FUNCTION_BLOCK "STD_LineSecStdSub2"	// FB 90
TITLE = Line and section control standard subroutines
//OPYRIGHT:    (C) 2000 BY  BUHLER LTD.
//                           CH-9240 UZWIL  SWITZERLAND
//
//PRODUCT:      STD_MU664    
//
//TITLE:        Line and section control standard subroutines
//              
//              Standardfunktionen für Linien und Sektionen              
//              
//
//--------------------------------------------------------------------------------
//
//IDENT:        AUTOR:              DEPT:                              DATE:
//
//STD_FB90.2.5  A. Egli             CT3                               11-Aug-2003
//              Sub2071: PICFU.SectionInfoCode     
//STD_FB90.2.4  Ph. Engler          MU664                             04-Aug-2003
//              Sub1061: LB not LW                    
//STD_FB90.2.3  Ph. Engler          MU664                             30-Aug-2003
//              Sub1061: Copy  #VarTemp.InOutValue3 to TmpDInt
//                       LB not LW                    
//STD_FB90.2.1  A.Egli              CT3                               14-Mai-2003
//              Sub1001: On Off Command Line
//STD_FB90.2.0  A.Egli              CT3                               18-Oct-2002
//              New release: Function moved from FC120 to FB90
//STD_FC120.1.12Ph. Engler          MU664                             23-Aug-2002
//              - Function (4,1) added: Search group manual mode
//STD_FC120.1.11Ph. Engler          MU664                              30-Apr-2002
//              - Function (1,55) and (2,55) modified: Stopping/Stopped
//STD_FC120.1.10Ph. Engler          MU664                              21-Mar-2002
//              - Function (2,55): starting until S.ToSSW.infStarted
//STD_FC120.1.9 Ph. Engler          MU664                              12-Mar-2002
//              Status codes for WinCoS implemented:
//              - General group colour code
//              - Line and Section info code
//STD_FC120.1.8 Ph. Engler          MU664                              20-Mar-2001
//              Line status colour for 2-4 section implemented
//STD_FC120.1.7 Ph. Engler          MU664                              20-Dec-2000
//              Pre stop weight for cmdSequenceStop
//STD_FC120.1.6 Ph. Engler          MU664                              14-Dec-2000
//              - Substitude BtmpInCode into recipe extended, tmpInCode 3 
//              - JS Job paramter flags (2,2) Sta-Address corrected
//STD_FC120.1.5 Ph. Engler          MU664                              01-Nov-2000
//              CmdSequenceStop only if section is in StActive           
//STD_FC120.1.4 Ph. Engler          MU664                              19-Okt-2000
//              Update SND-Binlist staSameSndRcv:
//               Suppression of the error meassage 'bin not found'
//STD_FC120.1.3 Ph. Engler          MU664                              28-Jun-2000
//              Section text and colour code extension 
//              with code 702, 703 and 1402
//STD_FC120.1.2 Ph. Engler          MU664                              04-May-2000
//              LS Line state/fault protocolling (1,10)
//               esXXX corrected 
//STD_FC120.1.1 Ph. Engler          MU664                              29-Mar-2000
//              Line log messages implemented
//STD_FC120.1.0 Ph. Engler          MU664                              05-Jan-2000
//              1st Release
//
//--------------------------------------------------------------------------------
//
//PURPOSE:      
//
//RESTRICTIONS:
//
//--------------------------------------------------------------------------------
//
AUTHOR : EA
FAMILY : STD
NAME : STD_FB90
VERSION : 2.5
VAR_INPUT
  InCode : INT ;
END_VAR
VAR
  Para : STRUCT
   ParSecNr : INT  := 1;
   ParLineDB_ParFirstSecDB : INT  := 320;
   spare4 : INT ;
   ParNextSecDB : INT ;	//Next section DB of this project line
   ParSecDataFirstByte : INT  := 240;
   ParSecDataLenNomValue : INT  := 20;
   ParSecDataLenAcValue : INT  := 20;
   ParBinDataFirstByte : INT  := 300;
   ParBinDataLength : INT  := 72;
  END_STRUCT ;
  VarTemp : STRUCT
   InOutValue1 : INT ;
   InOutValue2 : INT ;
   InOutValue3 : DINT ;
   InOutValue4 : DINT ;
   InOutValue5 : DINT ;
   InOutValue6 : DINT ;
  END_STRUCT ;
  ChangeBit : STRUCT
   spare : BYTE ;
   CBit1 : BOOL ;
   CBit2 : BOOL ;
   CBit3 : BOOL ;
   CBit4 : BOOL ;
  END_STRUCT ;
  ToASW : STRUCT
   spare00 : WORD ;
   CmdModify : BOOL ;
   CmdNewBatch : BOOL ;
   CmdDataMoved : BOOL ;
   InfSameJobPrevSec : BOOL ;
   InfSameJobNextSec : BOOL ;
   InfSameBatchPrevSec : BOOL ;
   InfSameBatchNextSec : BOOL ;
   InfSameJobLineDB : BOOL ;	//Job in reveive box is equal
   InfEmptyingTimeEnd : BOOL ;
   InfWayAdjustTimeEnd : BOOL ;
   spare32 : BOOL ;
   spare33 : BOOL ;
   spare34 : BOOL ;
   spare35 : BOOL ;
   spare36 : BOOL ;
   InfDataReady : BOOL ;
   Func : UDT 10601;
   Transition : STRUCT
    spare00 : BYTE ;
    ToPassive : BOOL ;
    ToWait : BOOL ;
    ToActive : BOOL ;
    ToReady : BOOL ;
    ToEmptying : BOOL ;
    ToEmptied : BOOL ;
    ToIdling : BOOL ;
   END_STRUCT ;
   spare10 : WORD ;
   spare12 : DWORD ;
   spare16 : DWORD ;
  END_STRUCT ;
  ToSSW : STRUCT
   InfStopped : BOOL ;
   spare01 : BOOL ;
   InfStarted : BOOL ;
   spare03 : BOOL ;
   spare04 : BOOL ;
   InfFeeding : BOOL ;
   spare06 : BOOL ;
   spare07 : BOOL ;
   spare00 : BOOL ;
   CmdGotoActive : BOOL ;
   CmdGotoReady : BOOL ;
   CmdGotoEmptying : BOOL ;
   CmdGotoEmptied : BOOL ;
   CmdGotoIdling : BOOL ;
   CmdGotoPassive : BOOL ;
   spare17 : BOOL ;
   InfReadyForNewBatch : BOOL ;
   CmdSendResult : BOOL ;
   InfPulseTimer : BOOL ;
   CmdNewWay : BOOL ;
   spare24 : BOOL ;
   spare25 : BOOL ;
   spare26 : BOOL ;
   InfReleaseEmptyingTime : BOOL ;
   Func : UDT 10601;
   InPrevSecDB : INT ;	//Previouse section DB in product flow
   InNextSecDB : INT ;	//Next section DB in product flow
   spare12 : DWORD ;
   spare16 : DWORD ;
  END_STRUCT ;
  PCWrite : STRUCT 	//PC Write : Section Data
   Hsk : STRUCT
    Q_Status : BOOL ;
    Q_Result : BOOL ;
    spare02 : BOOL ;
    spare03 : BOOL ;
    spare04 : BOOL ;
    spare05 : BOOL ;
    Q_MDEEData : BOOL ;	//Acknowledge data sended to MDEE by PCC
    Q_MYRAData : BOOL ;	//Acknowledge data sended to MYRA by PCC
    F_Define : BOOL ;
   END_STRUCT ;
   spare2 : WORD ;
   Func : UDT 10601;
   Value1 : INT ;
   Value2 : INT ;
   Value3 : INT ;
   ParWayAdjustTime : INT  := 2;
   Value5 : INT ;
   ParEmptyingTime : INT  := 20;
  END_STRUCT ;
  PCRead : STRUCT 	//PC Read : Section Data
   Hsk : STRUCT
    F_Status : BOOL ;
    F_Result : BOOL ;
    F_2 : BOOL ;
    F_3 : BOOL ;
    F_4 : BOOL ;
    F_5 : BOOL ;
    F_MDEEData : BOOL ;	//Request PCC to send data to MDEE
    F_MYRAData : BOOL ;	//Request PCC to send data to MYRA
   END_STRUCT ;
   ErrElement : INT ;
   ErrCode : INT ;
   ErrObject : INT ;	//(*new*)
   Step : STRUCT
    spare : BYTE ;
    StPassive : BOOL ;
    StWait : BOOL ;
    StActive : BOOL ;
    StReady : BOOL ;	//Line= Idling
    StEmptying : BOOL ;
    StEmptied : BOOL ;
    StIdling : BOOL ;
   END_STRUCT ;
   State : STRUCT
    spare : BYTE ;
    StStopped : BOOL ;
    StStarting : BOOL ;
    StStarted : BOOL ;
    StStopping : BOOL ;
    spare04 : BOOL ;
    StFeeding : BOOL ;
   END_STRUCT ;
   Fault : UDT 10602;
   Status : UDT 10603;
   StateColor : INT ;
   StateInfoCode : INT ;	//Line: GenGrpColorCode
   ExtStatus : INT ;
   OutWayAdjustTime_ExtOn : INT ;
   OutStartWarningTime : INT ;	//Copy of Startwarning modul
   OutEmptyingTime : INT ;
   Value7 : INT ;
   Value8 : INT ;
   Value9 : INT ;
   Value10 : INT ;
   Value11 : INT ;
   Value12 : INT ;
   Value13 : INT ;
   Value14 : INT ;
   Value15 : INT ;
   Value16 : INT ;
   Value17 : INT ;
   Value18 : INT ;
   Value19 : INT ;
  END_STRUCT ;
  JobNom : STRUCT 	//PC Read: Job header: Nominal values
   JobNr : DINT ;
   JobWeight : DINT ;	//Total Job weight
   BatchNo : INT  := 10;	//Number of batch requested form PC
   ScaleUsed : ARRAY  [1 .. 64 ] OF BOOL ;
   RecipeNr : INT ;
   BatchWeight : DINT ;
   BatchMinPpm : INT ;	//Minimum batch size [0.1%]
   BatchMaxPpm : INT ;	//Maximum batch size [0.1%]
   BatchNoOffset : INT ;	//Batch number of first batch
   MixingTime : INT ;	//Mixing time
   JobChangeTime : INT ;	//Job change time
   FeedingTime : INT ;	//Feeding Time
   Value13 : INT ;
   Value14 : INT ;
  END_STRUCT ;
  JobAc : STRUCT 	//PC Read: Job header: Actual values
   StaBatch : STRUCT
    spare0 : BOOL ;
    spare1 : BOOL ;
    spare2 : BOOL ;
    spare3 : BOOL ;
    spare4 : BOOL ;
    spare5 : BOOL ;
    StaEmptyingBatch : BOOL ;
    StaScaleRecipeValid : BOOL ;
    StaErrBatch : BOOL ;
    StaHandAddReady : BOOL ;
    StaRegistrated : BOOL ;
    StaLastBatch : BOOL ;
    StaDone : BOOL ;
   END_STRUCT ;
   JobWeight : DINT ;
   BatchNo : INT ;
   BatchNoCal : INT ;
   BatchWeightTarget : DINT ;	//Calculated target batch weight
   BatchWeightActual : DINT ;	//Actual weight of all dosed ingredient
   BatchSizePpm : INT ;	//Calculated batch size [1/1000]
   BatchValue8 : INT ;
   BatchValue9 : INT ;
   MixingTime : INT ;	//Mixing time
   JobChangeTime : INT ;	//Job change time
   FeedingTime : INT ;	//Feeding Time
   RecipePlace : INT ;	//Actual recipe place
   Value16 : INT ;
   Value17 : INT ;
   Value18 : INT ;
   Value19 : INT ;
  END_STRUCT ;
END_VAR
VAR_TEMP
  TmpWord : WORD ;
  TmpInt : INT ;
  TmpDInt : DINT ;
  TmpBool : BOOL ;
  tmpLineStStopped : BOOL ;
  tmpLineStaAutostart : BOOL ;
  tmpLineInfFeeding : BOOL ;
  DB9SecArray : DWORD ;	//Address Pointer Section in DB9
  tmpSecDB : INT ;
  tmpAddrGrInterfaceSec : DINT ;	//Pointer to Interface in section DB
  tmpLineDB : INT ;
  tmpRelevantGroups : DINT ;
  tmpSec_GenGrpCoulorCode : STRUCT
   lightGrey : BOOL ;
   Bit1 : BOOL ;
   darkGreen : BOOL ;
   magenta : BOOL ;
   red : BOOL ;
  END_STRUCT ;
  tmpLin_GenGrpCoulorCode : STRUCT
   lightGrey : BOOL ;
   Bit1 : BOOL ;
   darkGreen : BOOL ;
   magenta : BOOL ;
   red : BOOL ;
  END_STRUCT ;
  tmpStateColorS1 : STRUCT
   white : BOOL ;
   yellow : BOOL ;
   blue : BOOL ;
   dark_green : BOOL ;
   green : BOOL ;
   light_green : BOOL ;
   mangenta : BOOL ;
   red : BOOL ;
   Bit8 : BOOL ;
   Bit9 : BOOL ;
   Bit10 : BOOL ;
   Bit11 : BOOL ;
   Bit12 : BOOL ;
   brown : BOOL ;
   orange : BOOL ;
   tuerkis : BOOL ;
  END_STRUCT ;
  tmpStateColorS2 : STRUCT
   white : BOOL ;
   yellow : BOOL ;
   blue : BOOL ;
   dark_green : BOOL ;
   green : BOOL ;
   light_green : BOOL ;
   mangenta : BOOL ;
   red : BOOL ;
   Bit8 : BOOL ;
   Bit9 : BOOL ;
   Bit10 : BOOL ;
   Bit11 : BOOL ;
   Bit12 : BOOL ;
   brown : BOOL ;
   orange : BOOL ;
   tuerkis : BOOL ;
  END_STRUCT ;
  tmpStateColorS3 : STRUCT
   white : BOOL ;
   yellow : BOOL ;
   blue : BOOL ;
   dark_green : BOOL ;
   green : BOOL ;
   light_green : BOOL ;
   mangenta : BOOL ;
   red : BOOL ;
   Bit8 : BOOL ;
   Bit9 : BOOL ;
   Bit10 : BOOL ;
   Bit11 : BOOL ;
   Bit12 : BOOL ;
   brown : BOOL ;
   orange : BOOL ;
   tuerkis : BOOL ;
  END_STRUCT ;
  tmpStateColorS4 : STRUCT
   white : BOOL ;
   yellow : BOOL ;
   blue : BOOL ;
   dark_green : BOOL ;
   green : BOOL ;
   light_green : BOOL ;
   mangenta : BOOL ;
   red : BOOL ;
   Bit8 : BOOL ;
   Bit9 : BOOL ;
   Bit10 : BOOL ;
   Bit11 : BOOL ;
   Bit12 : BOOL ;
   brown : BOOL ;
   orange : BOOL ;
   tuerkis : BOOL ;
  END_STRUCT ;
  tmpStateColorLine : STRUCT
   white : BOOL ;
   yellow : BOOL ;
   blue : BOOL ;
   dark_green : BOOL ;
   green : BOOL ;
   light_green : BOOL ;
   mangenta : BOOL ;
   red : BOOL ;
   Bit8 : BOOL ;
   Bit9 : BOOL ;
   Bit10 : BOOL ;
   Bit11 : BOOL ;
   Bit12 : BOOL ;
   brown : BOOL ;
   orange : BOOL ;
   tuerkis : BOOL ;
  END_STRUCT ;
  tmpUserState : STRUCT 	//PIC FU
   stEmptying : BOOL ;
   stEmptied : BOOL ;
   stIdling : BOOL ;
   stFault : BOOL ;
   stHand : BOOL ;
   stHold : BOOL ;
   stStep : BOOL ;
   spare : BOOL ;
   stPassiv : BOOL ;
   stWait : BOOL ;
   stStarting : BOOL ;
   stStarted : BOOL ;
   stStopping : BOOL ;
   stStopped : BOOL ;
   stFeeding : BOOL ;
   stReady : BOOL ;
  END_STRUCT ;
END_VAR
BEGIN
NETWORK
TITLE = Init
      LAR2  P##InCode;
      L     DINO;
      T     #tmpLineDB;
      T     #tmpSecDB;
NETWORK
TITLE = Sub1001: LS Line On Off Command
//Called by line controler subroutines, with opened L-DB
      L     #InCode;
      L     1001;
      <>I;
      JC    LS01;
      L     #PCWrite.Value1;	// PCWrite.ExtFuncOn 
      T     #PCRead.OutWayAdjustTime_ExtOn;
//-Update ExtStatus------------------------
      L     #PCRead.ExtStatus;	// ExtStatus
      L     #PCWrite.Value1;	// PCWrite.ExtFuncOn 
      OD;	// 
      L     #PCWrite.Value2;	// PCWrite.ExtFuncOff 
      INVD;	//  
      AD;	//  
      T     #PCRead.ExtStatus;	//->ExtStatus
//Reset on commands 
      L     0;
      T     #PCWrite.Value1;	// PCWrite.ExtFuncOn 
//Reset off commands 
      L     0;
      T     #PCWrite.Value2;	// PCWrite.ExtFuncOff 
      BEU;
LS01: NOP   0;
NETWORK
TITLE = Sub1010: LS Line state/fault protocolling
//Called by line controler subroutines, with opened L-DB
//
//Output: LineDB.VarTemp.InOutValue1 = LineMsg
      L     #InCode;
      L     1010;
      <>I;
      JC    LS00;
//-Init var---
      L     0;
      T     MW 2018;
//Read old value: PCRead.StateColor
      L     #PCRead.StateColor;
      LAR1  P##tmpStateColorS1;	// LineDB.PCRead.StateColor
      T     LW [AR1,P#0.0];	//-->tmpStateColorS1
//-Generate summary step---
      A     #tmpStateColorS1.tuerkis;	// 
      =     M 2019.3;	// --> LineMsg.suspended
      SET;
      S     M 2019.0;	// --> LineMsg.terminated
      S     M 2019.1;	// --> LineMsg.stopped
      R     M 2019.2;	// --> LineMsg.started
      R     M 2019.4;	// --> LineMsg.faulted
      R     M 2019.5;	// --> LineMsg.warning
      R     M 2018.0;	// --> LineMsg.SenderEmpty
      R     M 2018.3;	// --> LineMsg.allPreselectRcvFull
      R     M 2018.4;	// --> LineMsg.MachinesNotAvailable
      L     #Para.ParLineDB_ParFirstSecDB;	// Para.ParFirstSecDB   
LOOP: T     #tmpSecDB;
      OPN   DI [#tmpSecDB];
      AN    #PCRead.Step.StPassive;	// Section
      AN    #PCRead.Step.StIdling;	// Section
      R     M 2019.0;	// --> LineMsg.terminated
      AN    #PCRead.State.StStopped;	// Section
      ON    #PCRead.Status.StaImmediateStopASW;	// Section
      R     M 2019.1;	// --> LineMsg.stopped
      AN    #PCRead.Step.StPassive;	// Section
      AN    #PCRead.Step.StIdling;	// Section
      S     M 2019.2;	// --> LineMsg.started
      A     #PCRead.Fault.EsMech;	// Section
      AN    #PCRead.Step.StPassive;	// Section
      AN    #PCRead.Step.StIdling;	// Section
      S     M 2019.4;	// --> LineMsg.faulted
      A     #PCRead.Fault.EsWarning;	// Section
      AN    #PCRead.Step.StPassive;	// Section
      AN    #PCRead.Step.StIdling;	// Section
      S     M 2019.5;	// --> LineMsg.warning
      A     #PCRead.Fault.EsEmpty;	// Section
      AN    #PCRead.Step.StPassive;	// Section
      AN    #PCRead.Step.StIdling;	// Section
      S     M 2018.0;	// --> LineMsg.SenderEmpty
      A     #PCRead.Fault.EsFull;	// Section
      AN    #PCRead.Step.StPassive;	// Section
      AN    #PCRead.Step.StIdling;	// Section
      S     M 2018.3;	// --> LineMsg.allPreselectRcvFull
      A     #PCRead.Fault.EsWayConflict;	// Section
      AN    #PCRead.Step.StPassive;	// Section
      AN    #PCRead.Step.StIdling;	// Section
      S     M 2018.4;	// --> LineMsg.MachinesNotAvailable
//-Check next section---
      L     0;
      L     #Para.ParNextSecDB;	// Section
      <>I;
      JC    LOOP;
//-Return messages---
      OPN   DI [#tmpLineDB];
      L     MW 2018;	// LineMsg
      T     #VarTemp.InOutValue1;
      BEU;
LS00: NOP   0;
NETWORK
TITLE = Sub1051: C1 Line status colour for 1 section
//Called by line controler subroutines
      L     #InCode;
      L     1051;
      <>I;
      JC    C100;
//Init
      L     0;
      LAR1  P##tmpStateColorLine;
      T     LW [AR1,P#0.0];	//-->tmpStateColorLine
//Read state of section 1
      L     #Para.ParLineDB_ParFirstSecDB;
      T     #tmpSecDB;
      OPN   DI [#tmpSecDB];	// Call 1st section
      L     #PCRead.StateColor;	// Section
      LAR1  P##tmpStateColorS1;
      T     LW [AR1,P#0.0];	//-->tmpStateColorS1
//-Red----------------------------------
      A     #tmpStateColorS1.red;	// Section
      S     #tmpStateColorLine.red;
      JC    C101;
//-Magenta------------------------------
      A     #tmpStateColorS1.mangenta;	// Section
      S     #tmpStateColorLine.mangenta;
      JC    C101;
//-Turkis-------------------------------
      A     #tmpStateColorS1.tuerkis;	// Section
      S     #tmpStateColorLine.tuerkis;
      JC    C101;
//-Brown--------------------------------
      A     #tmpStateColorS1.brown;	// Section
      S     #tmpStateColorLine.brown;
      JC    C101;
//-Orange-------------------------------
      A     #tmpStateColorS1.orange;	// Section
      S     #tmpStateColorLine.orange;
      JC    C101;
//-Lightgreen---------------------------
      A     #tmpStateColorS1.light_green;	// Section
      S     #tmpStateColorLine.light_green;
      JC    C101;
//-Green--------------------------------
      A     #tmpStateColorS1.green;	// Section
      S     #tmpStateColorLine.green;
      JC    C101;
//-Darkgreen----------------------------
      A     #tmpStateColorS1.dark_green;	// Section
      S     #tmpStateColorLine.dark_green;
      JC    C101;
//-Yellow-------------------------------
      A     #tmpStateColorS1.yellow;	// Section
      S     #tmpStateColorLine.yellow;
      JC    C101;
//-Blue---------------------------------
      A     #tmpStateColorS1.blue;	// Section
      S     #tmpStateColorLine.blue;
      JC    C101;
//-White--------------------------------
      A     #tmpStateColorS1.white;	// Section
      S     #tmpStateColorLine.white;	//(default)
//-Data to PCC--------------------------
C101: OPN   DI [#tmpLineDB];
      LAR1  P##tmpStateColorLine;
      L     LW [AR1,P#0.0];	// tmpStateColorLine
      L     #PCRead.StateColor;	// LineDB
      ==I;	// 
      BEC;
      S     #ChangeBit.CBit1;	// LineDB
      TAK;
      T     #PCRead.StateColor;	// LineDB
      BEU;
C100: NOP   0;
NETWORK
TITLE = Sub1052: C2 Line status colour for 2 section
//Called by line controler subroutines
//
//Inputs :
// no
//Outputs:
// no
//
      L     #InCode;
      L     1052;
      <>I;
      JC    C200;
//Init
      L     0;
      LAR1  P##tmpStateColorLine;
      T     LW [AR1,P#0.0];	//-->tmpStateColorLine
//Read Status Section 1
      L     #Para.ParLineDB_ParFirstSecDB;
      T     #tmpSecDB;
      OPN   DI [#tmpSecDB];	// Call 1st section DB Para.ParFirstSecDB
      L     #PCRead.StateColor;	// Section
      LAR1  P##tmpStateColorS1;
      T     LW [AR1,P#0.0];	//-->tmpStateColorS1
//Read Status Section2
      L     #Para.ParNextSecDB;	// Section
      T     #tmpSecDB;
      OPN   DI [#tmpSecDB];	// Call next section DB Para.ParNextSecDB
      L     #PCRead.StateColor;	// Section
      LAR1  P##tmpStateColorS2;
      T     LW [AR1,P#0.0];	//-->tmpStateColorS2
      OPN   DI [#tmpLineDB];	// Call line DB .Para.ParLineDB
//-Red----------------------------------
      A     #tmpStateColorS1.red;
      O     #tmpStateColorS2.red;
      S     #tmpStateColorLine.red;
      JC    C201;
//-Magenta------------------------------
      A     #tmpStateColorS1.mangenta;
      O     #tmpStateColorS2.mangenta;
      S     #tmpStateColorLine.mangenta;
      JC    C201;
//-Turkis-------------------------------
      A     #tmpStateColorS1.tuerkis;
      O     #tmpStateColorS2.tuerkis;
      S     #tmpStateColorLine.tuerkis;
      JC    C201;
//-Brown--------------------------------
      A     #tmpStateColorS1.brown;
      O     #tmpStateColorS2.brown;
      S     #tmpStateColorLine.brown;
      JC    C201;
//-Orange-------------------------------
      A     #tmpStateColorS1.orange;
      O     #tmpStateColorS2.orange;
      S     #tmpStateColorLine.orange;
      JC    C201;
//-Lightgreen---------------------------
      A     #tmpStateColorS1.light_green;
      O     #tmpStateColorS2.light_green;
      S     #tmpStateColorLine.light_green;
      JC    C201;
//-Green--------------------------------
      A     #tmpStateColorS1.green;
      O     #tmpStateColorS2.green;
      S     #tmpStateColorLine.green;
      JC    C201;
//-Darkgreen----------------------------
      A     #tmpStateColorS1.dark_green;
      O     #tmpStateColorS2.dark_green;
      S     #tmpStateColorLine.dark_green;
      JC    C201;
//-Blue---------------------------------
      A     #tmpStateColorS1.blue;
      O     #tmpStateColorS2.blue;
      S     #tmpStateColorLine.blue;
      JC    C201;
//-Yellow-------------------------------
      A     #tmpStateColorS1.yellow;
      O     #tmpStateColorS2.yellow;
      S     #tmpStateColorLine.yellow;
      JC    C201;
//-White--------------------------------
      A     #tmpStateColorS1.white;
      A     #tmpStateColorS2.white;
      S     #tmpStateColorLine.white;	// (default)
//-Data to PCC--------------------------
C201: OPN   DI [#tmpLineDB];
      LAR1  P##tmpStateColorLine;
      L     LW [AR1,P#0.0];	// tmpStateColorLine
      L     #PCRead.StateColor;	// LineDB
      ==I;
      BEC;
      S     #ChangeBit.CBit1;	// LineDB
      TAK;
      T     #PCRead.StateColor;	// LineDB
      BEU;
C200: NOP   0;
NETWORK
TITLE = Sub1053: C3 Line status colour for 3 section
//Called by line controler subroutines
//
//Inputs :
// no
//Outputs:
// no
//
      L     #InCode;
      L     1053;
      <>I;
      JC    C300;
//Init
      L     0;
      LAR1  P##tmpStateColorLine;
      T     LW [AR1,P#0.0];	//-->tmpStateColorLine
//Read Status Section1
      L     #Para.ParLineDB_ParFirstSecDB;
      T     #tmpSecDB;
      OPN   DI [#tmpSecDB];	// Call 1st section DB Para.ParFirstSecDB
      L     #PCRead.StateColor;	// Section
      LAR1  P##tmpStateColorS1;
      T     LW [AR1,P#0.0];	//-->tmpStateColorS1
//Read Status Section2
      L     #Para.ParNextSecDB;	// Section
      T     #tmpSecDB;
      OPN   DI [#tmpSecDB];	// Call next section DB Para.ParNextSecDB
      L     #PCRead.StateColor;	// Section
      LAR1  P##tmpStateColorS2;
      T     LW [AR1,P#0.0];	//-->tmpStateColorS2
//Read Status Section3
      L     #Para.ParNextSecDB;	// Section
      T     #tmpSecDB;
      OPN   DI [#tmpSecDB];	// Call next section DB Para.ParNextSecDB
      L     #PCRead.StateColor;	// Section
      LAR1  P##tmpStateColorS3;
      T     LW [AR1,P#0.0];	//-->tmpStateColorS3
//-Red----------------------------------
      OPN   DI [#tmpLineDB];
      A     #tmpStateColorS1.red;
      O     #tmpStateColorS2.red;
      O     #tmpStateColorS3.red;
      S     #tmpStateColorLine.red;
      JC    C301;
//-Magenta------------------------------
      A     #tmpStateColorS1.mangenta;
      O     #tmpStateColorS2.mangenta;
      O     #tmpStateColorS3.mangenta;
      S     #tmpStateColorLine.mangenta;
      JC    C301;
//-Turkis-------------------------------
      A     #tmpStateColorS1.tuerkis;
      O     #tmpStateColorS2.tuerkis;
      O     #tmpStateColorS3.tuerkis;
      S     #tmpStateColorLine.tuerkis;
      JC    C301;
//-Brown--------------------------------
      A     #tmpStateColorS1.brown;
      O     #tmpStateColorS2.brown;
      O     #tmpStateColorS3.brown;
      S     #tmpStateColorLine.brown;
      JC    C301;
//-Orange-------------------------------
      A     #tmpStateColorS1.orange;
      O     #tmpStateColorS2.orange;
      O     #tmpStateColorS3.orange;
      S     #tmpStateColorLine.orange;
      JC    C301;
//-Lightgreen---------------------------
      A     #tmpStateColorS1.light_green;
      O     #tmpStateColorS2.light_green;
      O     #tmpStateColorS3.light_green;
      S     #tmpStateColorLine.light_green;
      JC    C301;
//-Green--------------------------------
      A     #tmpStateColorS1.green;
      O     #tmpStateColorS2.green;
      O     #tmpStateColorS3.green;
      AN    #tmpStateColorS2.dark_green;
      S     #tmpStateColorLine.green;
      JC    C301;
//-Darkgreen----------------------------
//      U     #tmpStateColorS1.dark_green
      A     #tmpStateColorS2.dark_green;
//      U     #tmpStateColorS3.dark_green
      S     #tmpStateColorLine.dark_green;
      JC    C301;
//-Blue---------------------------------
      A     #tmpStateColorS1.blue;
      O     #tmpStateColorS2.blue;
      O     #tmpStateColorS3.blue;
      S     #tmpStateColorLine.blue;
      JC    C301;
//-Yellow-------------------------------
//      U     #tmpStateColorS1.yellow
      A     #tmpStateColorS2.yellow;
//      U     #tmpStateColorS3.yellow
      S     #tmpStateColorLine.yellow;
      JC    C301;
//-White--------------------------------
//      U     #tmpStateColorS1.white
      A     #tmpStateColorS2.white;
      A     #tmpStateColorS3.white;
      S     #tmpStateColorLine.white;	// (default)
      JC    C301;
//-Data to PCC--------------------------
C301: OPN   DI [#tmpLineDB];
      LAR1  P##tmpStateColorLine;
      L     LW [AR1,P#0.0];	// tmpStateColorLine
      L     #PCRead.StateColor;	// LineDB
      ==I;	// 
      BEC;
      S     #ChangeBit.CBit1;	// LineDB
      TAK;
      T     #PCRead.StateColor;	// LineDB
      BEU;
C300: NOP   0;
NETWORK
TITLE = Sub1054: C4 Line status colour for 4 section
//Called by line controler subroutines
      L     #InCode;
      L     1054;
      <>I;
      JC    C400;
//Init
      L     0;
      LAR1  P##tmpStateColorLine;
      T     LW [AR1,P#0.0];	//-->tmpStateColorLine
//Read Status Section1
      L     #Para.ParLineDB_ParFirstSecDB;
      T     #tmpSecDB;
      OPN   DI [#tmpSecDB];	// Call 1st section DB Para.ParFirstSecDB
      L     #PCRead.StateColor;	// Section
      LAR1  P##tmpStateColorS1;
      T     LW [AR1,P#0.0];	//-->tmpStateColorS1
//Read Status Section2
      L     #Para.ParNextSecDB;	// Section
      T     #tmpSecDB;
      OPN   DI [#tmpSecDB];	// Call next section DB Para.ParNextSecDB
      L     #PCRead.StateColor;	// Section
      LAR1  P##tmpStateColorS2;
      T     LW [AR1,P#0.0];	//-->tmpStateColorS2
//Read Status Section3
      L     #Para.ParNextSecDB;	// Section
      T     #tmpSecDB;
      OPN   DI [#tmpSecDB];	// Call next section DB Para.ParNextSecDB
      L     #PCRead.StateColor;	// Section
      LAR1  P##tmpStateColorS3;
      T     LW [AR1,P#0.0];	//-->tmpStateColorS3
//Read Status Section4
      L     #Para.ParNextSecDB;	// Section
      T     #tmpSecDB;
      OPN   DI [#tmpSecDB];	// Call next section DB Para.ParNextSecDB
      L     #PCRead.StateColor;	// Section
      LAR1  P##tmpStateColorS4;
      T     LW [AR1,P#0.0];	//-->tmpStateColorS4
      OPN   DI [#tmpLineDB];	// Call line DB 
// 
//-Red----------------------------------
      A     #tmpStateColorS1.red;
      O     #tmpStateColorS2.red;
      O     #tmpStateColorS3.red;
      O     #tmpStateColorS4.red;
      S     #tmpStateColorLine.red;
      JC    C401;
//-Magenta------------------------------
      A     #tmpStateColorS1.mangenta;
      O     #tmpStateColorS2.mangenta;
      O     #tmpStateColorS3.mangenta;
      O     #tmpStateColorS4.mangenta;
      S     #tmpStateColorLine.mangenta;
      JC    C401;
//-Turkis-------------------------------
      A     #tmpStateColorS1.tuerkis;
      O     #tmpStateColorS2.tuerkis;
      O     #tmpStateColorS3.tuerkis;
      O     #tmpStateColorS4.tuerkis;
      S     #tmpStateColorLine.tuerkis;
      JC    C401;
//-Yellow-------------------------------
      A     #tmpStateColorS1.yellow;
      A     #tmpStateColorS2.yellow;
      A     #tmpStateColorS3.yellow;
      A     #tmpStateColorS4.yellow;
      S     #tmpStateColorLine.yellow;
      JC    C401;
//-Brown--------------------------------
      A     #tmpStateColorS1.brown;
      O     #tmpStateColorS2.brown;
      O     #tmpStateColorS3.brown;
      O     #tmpStateColorS4.brown;
      S     #tmpStateColorLine.brown;
      JC    C401;
//-Orange-------------------------------
      A     #tmpStateColorS1.orange;
      O     #tmpStateColorS2.orange;
      O     #tmpStateColorS3.orange;
      O     #tmpStateColorS4.orange;
      S     #tmpStateColorLine.orange;
      JC    C401;
//-Lightgreen---------------------------
//      U     #tmpStateColorS1.light_green
//      U     #tmpStateColorS2.light_green
//      U     #tmpStateColorS3.light_green
//      U     #tmpStateColorS4.light_green
      CLR;
      S     #tmpStateColorLine.light_green;
      JC    C401;
//-Green--------------------------------
//      U     #tmpStateColorS1.green
//      U     #tmpStateColorS2.green
//      U     #tmpStateColorS3.green
//      U     #tmpStateColorS4.green
      CLR;
      S     #tmpStateColorLine.green;
      JC    C401;
//-Blue---------------------------------
      A     #tmpStateColorS1.white;
      A     #tmpStateColorS2.white;
      A     #tmpStateColorS3.white;
      A     #tmpStateColorS4.blue;
      S     #tmpStateColorLine.blue;
      JC    C401;
//-Darkgreen----------------------------
//      U     #tmpStateColorS1.dark_green
//      U     #tmpStateColorS2.dark_green
//      U     #tmpStateColorS3.dark_green
//      U     #tmpStateColorS4.dark_green
      A     #PCRead.Step.StActive;	// LineDB 
      O     #PCRead.Step.StReady;	// LineDB 
      S     #tmpStateColorLine.dark_green;
      JC    C401;
//-White--------------------------------
//      U     #tmpStateColorS1.white
//      U     #tmpStateColorS2.white
//      U     #tmpStateColorS3.white
//      U     #tmpStateColorS4.white
      A     #PCRead.Step.StPassive;	// LineDB
      O     #PCRead.Step.StIdling;	// LineDB
      S     #tmpStateColorLine.white;	// (default)
      JC    C401;
//-Data to PCC--------------------------
C401: OPN   DI [#tmpLineDB];
      LAR1  P##tmpStateColorLine;
      L     LW [AR1,P#0.0];	// tmpStateColorLine
      L     #PCRead.StateColor;	// LineDB
      ==I;	// 
      BEC;
      S     #ChangeBit.CBit1;	// LineDB
      TAK;
      T     #PCRead.StateColor;	// LineDB
      BEU;
C400: NOP   0;
NETWORK
TITLE = Sub1055: I1 Line info code for x sections WinCoS
      L     #InCode;
      L     1055;
      <>I;
      JC    I100;
// 
//-Begin-Scan all sections---
      L     #Para.ParLineDB_ParFirstSecDB;	// LineDB
      T     #tmpSecDB;
      OPN   DI [#tmpSecDB];	// Call Section DB
      SET;
      =     #tmpLineStaAutostart;
      =     #tmpLineStStopped;
      =     #tmpLineInfFeeding;
I1L1: AN    #PCRead.Status.StaAutostart;	// Section
      R     #tmpLineStaAutostart;
      AN    #PCRead.State.StStopped;	// Section
      AN    #PCRead.State.StStopping;	// Section
      R     #tmpLineStStopped;
      AN    #ToSSW.InfFeeding;	// Section
      R     #tmpLineInfFeeding;
//-End-Scan all sections--- 
      L     #Para.ParNextSecDB;	// Section
      L     0;
      <>I;
      JCN   I101;
      L     #Para.ParNextSecDB;
      T     #tmpSecDB;
      OPN   DI [#tmpSecDB];	// Call next S-DB
      JU    I1L1;
//-End-Scan all sections---
//===Line =============================================================
I101: OPN   DI [#tmpLineDB];	// Call L-DB
//=Build MainInfoCode=================
//-Fault------------------------------
      A     #PCRead.Fault.EsMech;	// LineDB
      O     #PCRead.Fault.EsDosing;	// LineDB
      O     #PCRead.Fault.EsBatchSize;	// LineDB
      O     #PCRead.Fault.EsRefillLevel;	// LineDB
      AN    #PCRead.Step.StPassive;	// LineDB
      AN    #PCRead.Step.StIdling;	// LineDB
      L     2#100000000000000;	// bit_main_status.passiv
      L     1500;	// code.Fault
      JC    I102;
//-Passive------------------------------
      A     #PCRead.Step.StPassive;	// LineDB
      L     2#1;	// bit_main_status.passiv
      L     100;	// code.st_passiv
      JC    I102;
//-AvailableTest------------------------
      A     #PCRead.Step.StActive;	// LineDB
      O     #PCRead.Step.StReady;	// LineDB
      A     #PCRead.Fault.EsWayConflict;	// LineDB
      L     2#100;	// bit_main_status.AvailableTest 
      L     300;	// code.st_AvailableTest
      JC    I102;
//-Stopped------------------------------
      A     #PCRead.Step.StActive;	// LineDB
      O     #PCRead.Step.StReady;	// LineDB
      A     #tmpLineStStopped;
      L     2#10000000000000;	// bit_main_status.stopped 
      L     1400;	// code.st_stopped
      JC    I102;
//-Suspended----------------------------
      A     #PCRead.Step.StActive;	// LineDB
      O     #PCRead.Step.StReady;	// LineDB
      AN    #tmpLineInfFeeding;
      L     2#100000;	// bit_main_status.suspended 
      L     600;	// code.st_suspended
      JC    I102;
//-Running------------------------------
      A     #PCRead.Step.StActive;	// LineDB
      O     #PCRead.Step.StReady;	// LineDB
      L     2#1000000;	// bit_main_status.running 
      L     700;	// code.st_running
      JC    I102;
//-Idling-------------------------------
      A     #PCRead.Step.StIdling;	// LineDB
      L     2#100000000000;	// bit_main_status.idling 
      L     1200;	// code.st_idling
      JC    I102;
//-No State-----------------------------
      L     2#0;	// bit_main_status.no_state 
      L     0;	// code.st_no_state
I102: T     #TmpInt;	// line text status
      TAK;
      T     #TmpWord;	// bit_main_status
// 
//=Build SubInfoCode====================
//-Fault--------------------------------
      OPN   DI [#tmpLineDB];
//-ReStart------------------------------
      L     #TmpWord;	// bit_main_status
      L     2#110000001100000;	// mask with restart code
      AW;
      JZ    I1N2;
      A     #PCRead.Status.StaImmediateStop;	// LineDB
      O     #PCRead.Status.StaTransferOff;	// LineDB
      O     #PCRead.Status.StaFeedOff;	// LineDB
      AN    #PCRead.Status.StaStep;	// LineDB
      ON    #tmpLineStaAutostart;
      L     3;	// code.restart
      JC    I103;
//-Step mode----------------------------
I1N2: L     #TmpWord;	// bit_main_status
      L     2#110000001101101;	// mask with step-mode code
      AW;
      JZ    I1N3;
      A     #PCRead.Status.StaStep;	// LineDB
      L     4;	// code.Step-mode
      JC    I103;
//-Hold---------------------------------
I1N3: L     #TmpWord;	// bit_main_status
      L     2#110100001101101;	// mask with step-mode code
      AW;
      JZ    I1N4;
      A     #PCRead.Status.StaHold;	// LineDB
      L     6;	// code.Step-mode
      JC    I103;
//-Warning------------------------------
I1N4: L     #TmpWord;	// bit_main_status
      L     2#110100001101000;	// mask with warning code
      AW;
      JZ    I1N5;
      A     #PCRead.Fault.EsWarning;	// LineDB
      L     1;	// code.Warning
      JC    I103;
//-Loaded-------------------------------
I1N5: L     #TmpWord;	// bit_main_status
      L     2#100000000001;	// mask with loaded code
      AW;
      JZ    I1N6;
      A     #PCRead.Status.StaLoaded;	// LineDB
      L     5;	// code.Loaded
      JC    I103;
//-NoSubState---------------------------
I1N6: L     0;	// code.NoSubState
// 
//=Build InfoCode=======================
I103: L     #TmpInt;	// MainInfoCode
      +I;	// Add SubInfoCode
      T     #PCRead.StateColor;	//-->LineDB
      BEU;
I100: NOP   0;
NETWORK
TITLE = Sub1061: GC GGRs status colour WinCoS
//Inputs :
// LineDB.VarTemp.InOutValue3 = Relevant Groups
//
//Outputs:
// no
//
      L     #InCode;
      L     1061;
      <>I;
      JC    GC00;
//-Init--- 
      L     #VarTemp.InOutValue3;	//[2.3]
      T     #TmpDInt;	//[2.3]
      L     0;
      LAR1  P##tmpLin_GenGrpCoulorCode;
      T     LW [AR1,P#0.0];	//Reset tmpLin_GenGrpCoulorCode
      OPN   "GCS7_GrCtrlDB";
//============================================
//Loop Section 
//============================================
      L     "GCS7_GrCtrlDB".ParByteNoSecDB;	//ParByteNoSecDB
      SLD   3;
GCLS: T     #DB9SecArray;
      OPN   "GCS7_GrCtrlDB";
//-----------------------------------
//Test End Of Array DB9.Sectio
      L     W#16#FFFF;
      L     DBW [#DB9SecArray];	// DB9.Section[x].DBNr
      ==I;
      JC    GCOT;	//-> Return
//-----------------------------------
//Read pointer to section interface
      T     #tmpSecDB;
      L     0;
      ==I;
      JC    GCNS;	//--> IF DBNr= 0 THEN  Next section
//-----------------------------------
//Start address Interface GroupControl in section
      LAR1  #DB9SecArray;
      OPN   "GCS7_GrCtrlDB";
      L     DBW [AR1,P#2.0];	//  DB9.Section[x].DBB
      SLD   3;
      T     #tmpAddrGrInterfaceSec;	//-->Pointer to instance in section DB
//-----------------------------------
//Check if section DB belongs to actual process line
      OPN   DI [#tmpSecDB];	// Call Section DB
      L     #Para.ParLineDB_ParFirstSecDB;	// S_DB
      L     #tmpLineDB;
      <>I;
      JC    GCNS;	//-->Next section
//-----------------------------------
//Start address Interface GroupControl in section
//========================================================= 
//Section[x]
//---------- 
//-Evaluate involved groups--- 
      LAR1  #tmpAddrGrInterfaceSec;	// Pointer to instance in section DB
      L     DID [AR1,P#52.0];	// SEC.Gr.OutSelected [08..01/16..09//24..17/32..25]
      L     #TmpDInt;	// USW selected relevant GGR [2.3]
      AD;
      T     #tmpRelevantGroups;	//--> Mask of relevant GGR
//-No State----------------------------------
      L     #tmpRelevantGroups;	// Mask of relevant GGR
      L     2#0;	// No group selected
      ==D;
      L     2#1;	// GenGrpStateCode.lightGrey (DB321.DBX x.0)
      JC    GC01;
//-Fault-------------------------------
      L     #tmpRelevantGroups;	// Mask of relevant GGR
      L     DB9.DBD 530;	// InFault [08..01/16..09//24..17/32..25]
      AD;
      L     0;
      <>D;
      L     2#10000;	// GenGrpStateCode.red (DB321.DBX x.4)
      JC    GC01;
//-Warning--------------------------------
      L     #tmpRelevantGroups;	// Mask of relevant GGR
      L     DB9.DBD 570;	// InWarning [08..01/16..09//24..17/32..25]
      AD;
      L     0;
      <>D;
      L     2#1000;	// GenGrpStateCode.magenta (DB321.DBX x.3)
      JC    GC01;
//-Else------------------------------
      L     2#100;	// GenGrpStateCode.darkGreen (DB321.DBX x.2)
GC01: LAR1  P##tmpSec_GenGrpCoulorCode;
      T     LB [AR1,P#0.0];	//-->tmpGenGrpCoulorCode  
//=================================================================
// Add Section-State to Line-State
//====================================================================
      OPN   DI [#tmpLineDB];	// Call L-DB
//-Fault--------------------------------
      A     #tmpLin_GenGrpCoulorCode.red;
      O     #tmpSec_GenGrpCoulorCode.red;
      L     2#10000;	// GenGrpCoulorCode.Fault 
      JC    GC02;
//-Warning------------------------------
      A     #tmpLin_GenGrpCoulorCode.magenta;
      O     #tmpSec_GenGrpCoulorCode.magenta;
      L     2#1000;	// GenGrpCoulorCode.Warning
      JC    GC02;
//-Started------------------------------
      A     #tmpLin_GenGrpCoulorCode.darkGreen;
      O     #tmpSec_GenGrpCoulorCode.darkGreen;
      L     2#100;	// GenGrpCoulorCode.Started
      JC    GC02;
//-No State-----------------------------
      L     2#1;	// GenGrpCoulorCode.lightGrey 
//-Save state---
GC02: LAR1  P##tmpLin_GenGrpCoulorCode;
      T     LB [AR1,P#0.0];	//Reset tmpLin_GenGrpCoulorCode //[2.4] LB not LW
//=== Call Next Section  =====================================
GCNS: L     #DB9SecArray;
      L     P#4.0;
      +D;	// Pointer to next section
      JU    GCLS;
GCOT: OPN   DI [#tmpLineDB];
      LAR1  P##tmpLin_GenGrpCoulorCode;
      L     LB [AR1,P#0.0];	//Reset tmpLin_GenGrpCoulorCode    //[2.4] LB not LW
      T     #PCRead.StateInfoCode;	//->LineDB  PCRead.GenGrpColorCode
GC00: NOP   0;
NETWORK
TITLE = Sub2001: SC Section commands
//Open DB = Section DB
//
//Inputs:
// SectionDB.VarTemp.InOutValue3 = Precutoff weight
      L     #InCode;
      L     2001;
      <>I;
      JC    SC00;
//--- FKT.immediate_stop---------------
      A     #PCRead.Status.StaHWStop;
      S     #ToSSW.Func.CmdImmediateStop;
//--- FKT.empty_section ---------------
      A     #JobAc.StaBatch.StaEmptyingBatch;
      S     #ToSSW.Func.CmdFeedOff;
      A     #JobAc.StaBatch.StaEmptyingBatch;
      A     #PCRead.Step.StActive;
      S     #ToSSW.Func.CmdSequenzStop;
      S     #PCRead.Status.StaLoaded;
//--- FKT.step_mode -------------------
      A     #PCRead.Status.StaStep;
      S     #ToSSW.Func.CmdFeedOff;
      A     #ToSSW.InfStarted;
      A     #PCRead.Step.StActive;
      S     #ToSSW.Func.CmdStepOff;
//--- FKT.sequnce_stop ----------------
      A(;
      L     #JobNom.FeedingTime;
      L     #JobAc.FeedingTime;
      <=I;
      A(;
      L     0;
      L     #JobNom.FeedingTime;
      <>I;
      );
      );
      O(;
      L     #JobNom.JobWeight;
      L     #VarTemp.InOutValue3;	// Prestop weight  [1.7]
      -D;	//                 [1.7]
      L     #JobAc.JobWeight;
      <=D;
      A(;
      L     0;
      L     #JobNom.JobWeight;
      <>D;
      );
      );
      A     #PCRead.Step.StActive;
      S     #ToSSW.Func.CmdSequenzStop;
      BEU;
SC00: NOP   0;
NETWORK
TITLE = Sub2003:SI Section init
//Called by section controler subroutines
//
//Open DB = Section DB
//
//Inputs :
// no
//Outputs:
// no
//
      L     #InCode;
      L     2003;
      <>I;
      JC    SI00;
//-FKT.immediate_stop------------------
      SET;
      R     #PCRead.Status.StaImmediateStop;
//-FKT.feeding_time--------------------
      L     0;
      T     #JobAc.FeedingTime;
      BEU;
SI00: NOP   0;
NETWORK
TITLE = Sub2004: FT Feeding time
//Called by section controler subroutines
//Open DB = Section DB
//
//Inputs :
// no
//Outputs:
// no
//
      L     #InCode;
      L     2004;
      <>I;
      JC    FT00;
      A     #PCRead.State.StFeeding;
      A     "SYS_Scan0_Tick1min";	//"SYS_Scan0_Tick1min"
      JCN   FT02;
      L     32767;
      L     #JobAc.FeedingTime;
      <=I;
      JC    FT01;	//If Time = maxValue then set to 0
      +     1;
      T     #JobAc.FeedingTime;
      BEU;
FT01: L     1;
      T     #JobAc.FeedingTime;
FT02: BEU;
FT00: NOP   0;
NETWORK
TITLE = Sub2051: ST Section status text and colour
//Called by section controler subroutines
//Open DB = Section DB
//
//Inputs :
// no
//Outputs:
// no
//
      L     #InCode;
      L     2051;
      <>I;
      JC    ST00;
//=Build auxiliary status===============
//-Passive------------------------------
      A     #PCRead.Step.StPassive;
      L     2#1;
      L     100;	// code.st_passiv
      JC    ST01;
//-Ready--------------------------------
      A     "SYS_infLog0";	// !! not used !!
      L     2#10;
      L     200;	// code.st_ready
      JC    ST01;
//-Available test-----------------------
      A     #PCRead.Step.StWait;
      L     2#100;
      L     300;	// code.st_available_test
      JC    ST01;
//-Start Warning------------------------
      A     #PCRead.Status.StaStartwarning;
      L     2#1000;
      L     400;	// code.st_startwarning
      JC    ST01;
//-Starting-----------------------------
      A     #PCRead.Step.StActive;
      A     #PCRead.State.StStarting;
      L     2#10000;
      L     500;	// code.st_starting
      JC    ST01;
//-Suspended----------------------------
      A     #PCRead.Step.StActive;
      A     #PCRead.State.StStarted;
      AN    #PCRead.State.StFeeding;
      L     2#100000;
      L     600;	// code.st_suspended
      JC    ST01;
//-Running------------------------------
      A     #PCRead.Step.StActive;
      A     #PCRead.State.StFeeding;
      L     2#1000000;
      L     700;	// code.st_running
      JC    ST01;
//-Wait---------------------------------
      A     #PCRead.Step.StReady;
      AN    #PCRead.Step.StEmptying;
      L     2#10000000;
      L     800;	// code.st_wait
      JC    ST01;
//-Emptying-----------------------------
      A     #PCRead.Step.StEmptying;
      AN    #ToSSW.InfReleaseEmptyingTime;
      AN    #PCRead.State.StStopped;
      L     2#100000000;
      L     900;	// code.st_emtying
      JC    ST01;
//-Emptying active----------------------
      A     #PCRead.Step.StEmptying;
      A     #ToSSW.InfReleaseEmptyingTime;
      AN    #PCRead.State.StStopped;
      L     2#1000000000;
      L     1000;	// code.st_emptying_activ
      JC    ST01;
//-Registration-------------------------
      A     #PCRead.Step.StEmptied;
      L     2#10000000000;
      L     1100;	// code.st_registration
      JC    ST01;
//-Idling-------------------------------
      A     #PCRead.Step.StIdling;
      L     2#100000000000;
      L     1200;	// code.st_idling
      JC    ST01;
//-Stopping-----------------------------
      A     #PCRead.State.StStopping;
      L     2#1000000000000;
      L     1300;	// code.st_stopping
      JC    ST01;
//-Stopped------------------------------
      AN    #PCRead.Step.StPassive;
      A     #PCRead.State.StStopped;
      L     2#10000000000000;
      L     1400;	// code.st_stopped
      JC    ST01;
//-No State-----------------------------
      L     2#0;
      L     0;	// code.st_no_state
ST01: T     #TmpInt;
      TAK;
      T     #TmpWord;
//==Status text=========================
//-Fault--------------------------------
      L     #TmpWord;
      L     2#11011111111100;	// status with fault code
      AW;
      JZ    ST11;
      A     #PCRead.Fault.EsMech;
      L     2;	// code.st_fault
      JC    ST02;
//-Warning------------------------------
ST11: L     #TmpWord;
      L     2#11011111111000;	// status with warning code
      AW;
      JZ    ST12;
      A     #PCRead.Fault.EsWarning;
      L     1;	// code.st_warning
      JC    ST02;
//-Restart------------------------------
ST12: L     #TmpWord;
      L     2#11000011110000;	// status with restart code
      AW;
      JZ    ST13;
      AN    #PCRead.Status.StaAutostart;
      L     3;	// code.st_restart
      JC    ST02;
//-Step mode----------------------------
ST13: L     #TmpWord;
      L     2#11000000111111;	// status with step_mode code
      AW;
      JZ    ST14;
      A     #PCRead.Status.StaStep;
      L     4;	// code.st_step_mode
      JC    ST02;
//-Loaded-------------------------------
ST14: L     #TmpWord;
      L     2#11000000000001;	// status with loaded code
      AW;
      JZ    ST15;
      A     #PCRead.Status.StaLoaded;
      L     5;	// code.st_loaded
      JC    ST02;
//-Mixing-------------------------------
ST15: L     #TmpWord;
      L     2#100000;	// status with mixing code
      AW;
      JZ    ST03;
      A     "SYS_infLog0";	// !!! not used !!!
      L     6;	// code.st_mixing
      JC    ST02;
      JU    ST03;
//-Build real text status---------------
ST02: L     #TmpInt;
      +I;
      T     #TmpInt;
//==Status colour=======================
//-Fault--------------------------------
ST03: L     #TmpWord;
      L     2#11011111111100;	// mask text code
      AW;
      JZ    ST31;
      A     #PCRead.Fault.EsMech;
      O     #PCRead.Fault.EsDosing;
      L     2#1000000000000000;	// additional_code.red
      JC    ST04;
//-Warning------------------------------
ST31: L     #TmpWord;
      L     2#11011111111000;	// mask text code
      AW;
      JZ    ST32;
      A     #PCRead.Fault.EsWarning;
      L     2#100000000000000;	// additional_code.magenta
      JC    ST04;
//-Ready for restart--------------------
ST32: L     #TmpWord;
      L     2#11011111111000;	// mask text code
      AW;
      JZ    ST33;
      A(;
      O     #PCRead.Step.StActive;
      O     #PCRead.Step.StReady;
      O     #PCRead.Step.StEmptying;
      O     #PCRead.Step.StEmptied;
      );
      AN    #PCRead.Status.StaAutostart;
      O;
      A     #PCRead.Status.StaFeedOff;
      A     #PCRead.Step.StActive;
      A     #PCRead.State.StStarted;
      AN    #PCRead.State.StFeeding;
      L     2#10000000;	// additional_code.tuerkis
      JC    ST04;
//-Step mode----------------------------
ST33: L     #TmpWord;
      L     2#11000000111111;	// mask text code
      AW;
      JZ    ST34;
      AN    #PCRead.Step.StPassive;
      A     #PCRead.Status.StaStep;
      L     2#100000;	// additional_code.brown
      JC    ST04;
//-Occupied-----------------------------
ST34: L     #TmpWord;
      L     2#100000000001;	// mask text code
      AW;
      JZ    ST35;
      A     #PCRead.Status.StaLoaded;
      L     2#1000000;	// additional_code.orange
      JC    ST04;
//-Starting-----------------------------
ST35: L     #TmpWord;
      L     2#11100;	// mask text code
      AW;
      JZ    ST36;
      L     2#10000000000000;	// code.light green
      JU    ST04;
//-Suspended----------------------------
ST36: L     #TmpWord;
      L     2#10100000;	// mask text code
      AW;
      JZ    ST37;
      L     2#1000000000000;	// code.green
      JU    ST04;
//-Running------------------------------
ST37: L     #TmpWord;
      L     2#1000000;	// mask text code
      AW;
      JZ    ST38;
      L     2#100000000000;	// code.dark green
      JU    ST04;
//-Emptying/Emptied---------------------
ST38: L     #TmpWord;
      L     2#11100000010;	// mask text code
      AW;
      JZ    ST39;
      L     2#10000000000;	// code.blue
      JU    ST04;
//-Stopping/Stopped---------------------
ST39: L     #TmpWord;
      L     2#11000000000000;	// mask text code
      AW;
      JZ    ST40;
      L     2#1000000000;	// code.yellow
      JU    ST04;
//-Passive/Idling-----------------------
ST40: L     #TmpWord;
      L     2#100000000001;	// mask text code
      AW;
      JZ    ST41;
      L     2#100000000;	// code.white
      JU    ST04;
//-Default------------------------------
ST41: L     2#100000000;	// code.weiss (default)
//=Data to MELE=========================
ST04: T     #TmpWord;	// --> Section colour state
//Check if any value changed PCRead.LineInfoCode
      L     #PCRead.StateColor;
      ==I;
      A(;
      L     #TmpInt;
      L     #PCRead.StateInfoCode;
      ==I;
      );
      BEC;
      S     #ChangeBit.CBit1;
      L     #TmpWord;	// Save section color status    
      T     #PCRead.StateColor;
      L     #TmpInt;	// Save section text status
      T     #PCRead.StateInfoCode;
      BEU;
ST00: NOP   0;
NETWORK
TITLE = Sub2055: SI Section info code : WinCoS
//Called by section controler subroutines
//
//Open DB = Section DB
//Inputs :
// no
//Outputs:
// no
//
      L     #InCode;
      L     2055;
      <>I;
      JC    I200;
// 
//=Build MainInfoCode===================
//-Fault--------------------------------
      A     #PCRead.Fault.EsMech;
      O     #PCRead.Fault.EsDosing;
      O     #PCRead.Fault.EsBatchSize;
      O     #PCRead.Fault.EsRefillLevel;
      AN    #PCRead.Step.StPassive;
      AN    #PCRead.Step.StIdling;
      L     2#100000000000000;
      L     1500;	// code.st_fault
      JC    I201;
//-Passive------------------------------
      A     #PCRead.Step.StPassive;
      L     2#1;
      L     100;	// code.st_passiv
      JC    I201;
//-Ready--------------------------------
      CLR;	// !! not used !!
      L     2#10;
      L     200;	// code.st_ready
      JC    I201;
//-Available test-----------------------
      A     #PCRead.Step.StWait;
      L     2#100;
      L     300;	// code.st_available_test
      JC    I201;
//-Start Warning------------------------
      A     #PCRead.Status.StaStartwarning;	// S.PCRead.Status.StaStartwarning
      L     2#1000;
      L     400;	// code.st_startwarning
      JC    I201;
//-Starting-----------------------------
      A     #PCRead.Step.StActive;
      AN    #ToSSW.InfStarted;
      AN    #PCRead.State.StStopped;
      AN    #PCRead.State.StStopping;
//    U     PCRead.State.StStarting    
      L     2#10000;
      L     500;	// code.st_starting
      JC    I201;
//-Suspended----------------------------
      A     #PCRead.Step.StActive;
      A     #PCRead.State.StStarted;
      AN    #PCRead.State.StFeeding;
      L     2#100000;
      L     600;	// code.st_suspended
      JC    I201;
//-Running------------------------------
      A     #PCRead.Step.StActive;
      A     #PCRead.State.StFeeding;
      L     2#1000000;
      L     700;	// code.st_running
      JC    I201;
//-Wait---------------------------------
      A     #PCRead.Step.StReady;
      AN    #PCRead.Step.StEmptying;
      L     2#10000000;
      L     800;	// code.st_wait
      JC    I201;
//-Emptying-----------------------------
      A     #PCRead.Step.StEmptying;
      AN    #ToSSW.InfReleaseEmptyingTime;
      AN    #PCRead.State.StStopped;
      L     2#100000000;
      L     900;	// code.st_emtying
      JC    I201;
//-Emptying active----------------------
      A     #PCRead.Step.StEmptying;
      A     #ToSSW.InfReleaseEmptyingTime;
      AN    #PCRead.State.StStopped;
      L     2#1000000000;
      L     1000;	// code.st_emptying_activ
      JC    I201;
//-Registration-------------------------
      A     #PCRead.Step.StEmptied;
      L     2#10000000000;
      L     1100;	// code.st_registration
      JC    I201;
//-Idling-------------------------------
      A     #PCRead.Step.StIdling;
      L     2#100000000000;
      L     1200;	// code.st_idling
      JC    I201;
//-Stopping-----------------------------
      A     #PCRead.State.StStopping;
      L     2#1000000000000;
      L     1300;	// code.st_stopping
      JC    I201;
//-Stopped------------------------------
      AN    #PCRead.Step.StPassive;
      A     #PCRead.State.StStopped;
      L     2#10000000000000;
      L     1400;	// code.st_stopped
      JC    I201;
//-No State-----------------------------
      L     2#0;
      L     0;	// code.st_no_state
I201: T     #TmpInt;
      TAK;
      T     #TmpWord;
//=Build SubInfoCode====================
//-Fault--------------------------------
//-Restart------------------------------
      L     #TmpWord;
      L     2#111011111111000;	// status with restart code
      AW;
      JZ    I212;
      A     #PCRead.Status.StaImmediateStop;
      O     #PCRead.Status.StaTransferOff;
      O     #PCRead.Status.StaFeedOff;
      AN    #PCRead.Status.StaStep;
      ON    #PCRead.Status.StaAutostart;
      L     3;	// code.st_restart
      JC    I202;
//-Step mode----------------------------
I212: L     #TmpWord;
      L     2#111000000111111;	// status with step_mode code
      AW;
      JZ    I213;
      A     #PCRead.Status.StaStep;
      L     4;	// code.st_step_mode
      JC    I202;
//-Hold---------------------------------
I213: L     #TmpWord;
      L     2#111100001111111;	// status with step_mode code
      AW;
      JZ    I214;
      A     #PCRead.Status.StaHold;
      L     6;	// code.st_step_mode
      JC    I202;
//-Warning------------------------------
I214: L     #TmpWord;
      L     2#111011111111000;	// status with warning code
      AW;
      JZ    I215;
      A     #PCRead.Fault.EsWarning;
      L     1;	// code.st_warning
      JC    I202;
//-Loaded-------------------------------
I215: L     #TmpWord;
      L     2#100000000001;	// status with loaded code
      AW;
      JZ    I216;
      A     #PCRead.Status.StaLoaded;	// S.PCRead.Status.StaLoaded
      L     5;	// code.st_loaded
      JC    I202;
//-NoSubState---------------------------
I216: L     0;	// code.NoSubState
// 
//=Build InfoCode=======================
I202: L     #TmpInt;	// MainInfoCode
      +I;	// Add SubInfoCode
      T     #PCRead.StateColor;
      BEU;
I200: NOP   0;
NETWORK
TITLE = Sub2071: PIC FU: Section info code
//Called by section controler subroutines
//
//Open DB = Section DB
//Inputs :
// no
//Outputs:
// no
//
      L     #InCode;
      L     2071;
      <>I;
      JC    I300;
// Reset 
      L     0;
      LAR1  P##tmpUserState;
      T     LW [AR1,P#0.0];
//-StFault
      A(;
      O     #PCRead.Fault.EsEmpty;
      O     #PCRead.Fault.EsFull;
      AN    #PCRead.Step.StPassive;
      AN    #PCRead.Step.StEmptying;
      AN    #PCRead.Step.StEmptied;
      AN    #PCRead.Step.StIdling;
      );
      O     #PCRead.Fault.EsWayConflict;
      O     #PCRead.Fault.EsMech;
      O     #PCRead.Fault.EsDosing;
      O     #PCRead.Fault.EsInterrupt;
      O     #PCRead.Fault.EsBatchSize;
      =     #tmpUserState.stFault;
      JC    Tran;
//-StPassive
      A     #PCRead.Step.StPassive;
      A     #PCRead.State.StStopped;
      AN    #PCRead.Status.StaHold;
      AN    #PCRead.Status.StaHand;
      AN    #PCRead.Status.StaStep;
      =     #tmpUserState.stPassiv;
      JC    Tran;
//-StWait
      A     #PCRead.Step.StWait;
      AN    #PCRead.Status.StaHold;
      AN    #PCRead.Status.StaHand;
      AN    #PCRead.Status.StaStep;
      =     #tmpUserState.stWait;
      JC    Tran;
//-StStarting--
      A     #PCRead.Step.StActive;
      A     #PCRead.State.StStarting;
      AN    #PCRead.Status.StaHold;
      AN    #PCRead.Status.StaHand;
      AN    #PCRead.Status.StaStep;
      =     #tmpUserState.stStarting;
      JC    Tran;
//-StStarted--
      A     #PCRead.Step.StActive;
      A     #PCRead.State.StStarted;
      AN    #PCRead.Status.StaHold;
      AN    #PCRead.Status.StaHand;
      AN    #PCRead.Status.StaStep;
      =     #tmpUserState.stStarted;
      JC    Tran;
//-StStopping--
      A     #PCRead.Step.StActive;
      A     #PCRead.State.StStopping;
      AN    #PCRead.Status.StaHold;
      AN    #PCRead.Status.StaHand;
      AN    #PCRead.Status.StaStep;
      =     #tmpUserState.stStopping;
      JC    Tran;
//-StStopped--
      A     #PCRead.Step.StActive;
      A     #PCRead.State.StStopped;
      AN    #PCRead.Status.StaHold;
      AN    #PCRead.Status.StaHand;
      AN    #PCRead.Status.StaStep;
      =     #tmpUserState.stStopped;
      JC    Tran;
//-StFeeding--
      A     #PCRead.Step.StActive;
      A     #PCRead.State.StFeeding;
      AN    #PCRead.Status.StaHold;
      AN    #PCRead.Status.StaHand;
      AN    #PCRead.Status.StaStep;
      AN    #PCRead.Status.StaEndOfJob;
      =     #tmpUserState.stFeeding;
      JC    Tran;
//-StReady--
      A     #PCRead.Step.StReady;
      AN    #PCRead.Status.StaHold;
      AN    #PCRead.Status.StaHand;
      AN    #PCRead.Status.StaStep;
      =     #tmpUserState.stReady;
      JC    Tran;
//-StEmptying--
      A     #PCRead.State.StFeeding;
      A     #PCRead.Status.StaEndOfJob;
      O     #PCRead.Step.StEmptying;
      AN    #PCRead.Status.StaHold;
      AN    #PCRead.Status.StaHand;
      AN    #PCRead.Status.StaStep;
      =     #tmpUserState.stEmptying;
      JC    Tran;
//-StEmptied--
      A     #PCRead.Step.StEmptied;
      AN    #PCRead.Status.StaHold;
      AN    #PCRead.Status.StaHand;
      AN    #PCRead.Status.StaStep;
      =     #tmpUserState.stEmptied;
      JC    Tran;
//-StIdling--
      A     #PCRead.Step.StIdling;
      AN    #PCRead.Status.StaHold;
      AN    #PCRead.Status.StaHand;
      AN    #PCRead.Status.StaStep;
      =     #tmpUserState.stIdling;
//-StHand--
      A     #PCRead.Status.StaHand;
      AN    #PCRead.Status.StaHold;
      AN    #PCRead.Status.StaStep;
      =     #tmpUserState.stHand;
      JC    Tran;
//-StHold--
      A     #PCRead.Status.StaHold;
      AN    #PCRead.Status.StaHand;
      AN    #PCRead.Status.StaStep;
      =     #tmpUserState.stHold;
      JC    Tran;
//-StStep--
      A     #PCRead.Status.StaStep;
      AN    #PCRead.Status.StaHold;
      AN    #PCRead.Status.StaHand;
      =     #tmpUserState.stStep;
      JC    Tran;
//Store New Code
Tran: L     #PCRead.StateInfoCode;
      LAR1  P##tmpUserState;
      L     LW [AR1,P#0.0];
      T     #PCRead.StateInfoCode;
// Changebit
      <>I;
      S     #ChangeBit.CBit1;
      BEU;
I300: NOP   0;
NETWORK
TITLE = End of block
      BE;
END_FUNCTION_BLOCK

FUNCTION_BLOCK "SYS_DPMultiDPInfo"	// FB 98
TITLE = Simple DP-Diagnostic
//
//COPYRIGHT:    (C) 1999  BUHLER AG, CH-9240 UZWIL, SWITZERLAND
//
//PRODUCT:      GCS7
//
//TITLE:        Simple DP-Diagnostic
//
//-------------------------------------------------------------------------
//
//IDENT:        AUTHOR:             DEPT:                       DATE:
//
//FB98.1.0      S. Kalberer         CT3                         15.12.1999
//              Adapted for more than 1 mastersystem from FC98.1A
//              
//-------------------------------------------------------------------------
//
//PURPOSE:      MANUAL : see Siemens manual DIAG21_d.PDF
//RESTRICTIONS: S7 type: see also Siemens manual
//
//-------------------------------------------------------------------------
//Input Parameters:
//-----------------
//
// InEnableCheck: 
//                FALSE = DP-Diagnostic check inactive
//                TRUE  = DP-Diagnostic check active
// InExtDPInterface (only relevant for S7-400):
//                FALSE = S7-300/ Internal Master DP-Interface (Master-CPU)
//                TRUE  = External Master DP-Interface  (CP, IM)
// InDPMasterSystemNo:
//                Number of DP-Mastersystems that was projected with STEP 7
//                (1= standard)
AUTHOR : SK
FAMILY : DP
NAME : MultiDP
VERSION : 1.0
VAR_INPUT
  InEnableCheck : BOOL ;	//Signal to enable the diagnostic check
  InExtDPInterface : BOOL ;	//only S7-400: 0= integrated (Master-CPU), 1= external (CP, IM)
  InDPMasterSystemNo : INT ;	//DP-Master System Number (projected with STEP 7)
END_VAR
VAR
  tmpDataField : ARRAY  [1 .. 50 ] OF //Internal used (not relevant for user)
  BYTE ;
  Sum_SlavesNotPresent : INT ;	//Summary slaves not present
  List_SlavesNotPresent : ARRAY  [1 .. 128 ] OF //List slaves not present
  BOOL ;
  Sum_SlavesError : INT ;	//Summary slaves with error
  List_SlavesError : ARRAY  [1 .. 128 ] OF //List slaves with error
  BOOL ;
  OutRetVal : INT ;	//Error return value
  OutBusy : BOOL ;	//Diagnostic check active
END_VAR
BEGIN
NETWORK
TITLE = Call Siemens FC 99 (GLOBAL_DP_INFO)
      CALL  "SIEMENS_GlobalDPInfo" (
           $1                       := #InEnableCheck,
           $2                       := #InExtDPInterface,
           $3                       := #InDPMasterSystemNo,
           $4                       := #tmpDataField,
           $5                       := #Sum_SlavesNotPresent,
           $6                       := #List_SlavesNotPresent,
           $7                       := #Sum_SlavesError,
           $8                       := #List_SlavesError,
           $9                       := #OutRetVal,
           $10                      := #OutBusy);
END_FUNCTION_BLOCK

FUNCTION_BLOCK "GCS7_StartWarning"	// FB 100
TITLE = StartWarning
//  
//COPYRIGHT:    (C) 2002  BUHLER AG, CH-9240 UZWIL,  SWITZERLAND
//
//PRODUCT:      GCS90
//
//TITLE:        FB 100 StartWarning 
// 
//-------------------------------------------------------------------------
//
//IDENT:        AUTHOR:             DEPT:                       DATE:
//
//FB100.1.2     A.Egli              CT3                        09-Mar-2004
//              Store Group DBNO of last warning 
//FB100.1.1     A.Egli              CT3                        21-Aug-2003
//              1st Release in S7
//FB100.1.0     A.Egli              CT3                         1-Jul-2002
//              1st Release in S7
//
//-------------------------------------------------------------------------
//
//PURPOSE:      MANUAL : see [LL.M4IxxMAN]
//
//RESTRICTIONS: S7
//
//
//-------------------------------------------------------------------------
//
AUTHOR : EA
FAMILY : GCS7LL
NAME : StartWa
VERSION : 1.2
VAR_INPUT
  InModeHigher : BOOL ;	//Higher    security : Every start
  InArea : INT ;
  InEnable : BOOL ;
  InLocal : BOOL ;
  InStarted : BOOL ;
  InCmdNext : BOOL ;
END_VAR
VAR_OUTPUT
  OutCmdNext : BOOL ;
  OutStartwarning : BOOL ;
END_VAR
VAR
  ParStartwarningTime : INT  := 10;	//[s]
  ParStartReleaseTimeL : INT  := 32767;	//[s] Low  security
  ParStartReleaseTimeH : INT  := 30;	//[s] High security
  ParRequestTime : INT  := 10;	//[0.1s]
  OutWarningObjectDB : INT ;	//Last Group DB how has run Startwarning
  OutWarningArea : INT ;	//Last Area how has run the Startwarning
  Spare2 : INT ;
  Spare3 : INT ;
  Spare4 : INT ;
  Area : ARRAY  [0 .. 20 ] OF STRUCT
   OutStartwarningRunning : BOOL ;
   OutStartReleaseRunningL : BOOL ;
   OutStartReleaseRunningH : BOOL ;
   CmdStartStartWarning : BOOL ;
   CmdResetStartWarning : BOOL ;
   tmpFlag200ms : BOOL ;	//flag of 200ms tag
   tmpFlag1s : BOOL ;	//flag of 1 s tag
   OutRequestTime : INT ;	//[0.1s]
   OutStartwarningTime : INT ;	//[s]
   OutStartReleaseTimeL : INT ;	//[s]
   OutStartReleaseTimeH : INT ;	//[s]
  END_STRUCT ;
  TmpArea : STRUCT
   OutStartwarningRunning : BOOL ;
   OutStartReleaseRunningL : BOOL ;
   OutStartReleaseRunningH : BOOL ;
   CmdStartStartWarning : BOOL ;
   CmdResetStartWarning : BOOL ;
   tmpFlag200ms : BOOL ;	//flag of 200ms tag
   tmpFlag1s : BOOL ;	//flag of 1 s tag
   OutRequestTime : INT ;	//[0.1s]
   OutStartwarningTime : INT ;	//[s]
   OutStartReleaseTimeL : INT ;	//[s]
   OutStartReleaseTimeH : INT ;	//[s]
  END_STRUCT ;
  TmpEnd : INT ;
END_VAR
VAR_TEMP
  AddrReading : DINT ;
  tmpLenArea : DINT ;
END_VAR
BEGIN
NETWORK
TITLE = Read Area Data
      L     #InArea;
      L     20;
      >I;
      BEC;
      L     P##TmpEnd;
      L     P##TmpArea;
      -D;
      T     #tmpLenArea;
      L     #InArea;
      *D;
      L     P##Area;
      +D;
      T     #AddrReading;
//====================================
      LAR1  #AddrReading;
      L     DID [AR1,P#0.0];
      LAR1  P##TmpArea;
      T     DID [AR1,P#0.0];
      LAR1  #AddrReading;
      L     DID [AR1,P#4.0];
      LAR1  P##TmpArea;
      T     DID [AR1,P#4.0];
      LAR1  #AddrReading;
      L     DIW [AR1,P#8.0];
      LAR1  P##TmpArea;
      T     DIW [AR1,P#8.0];
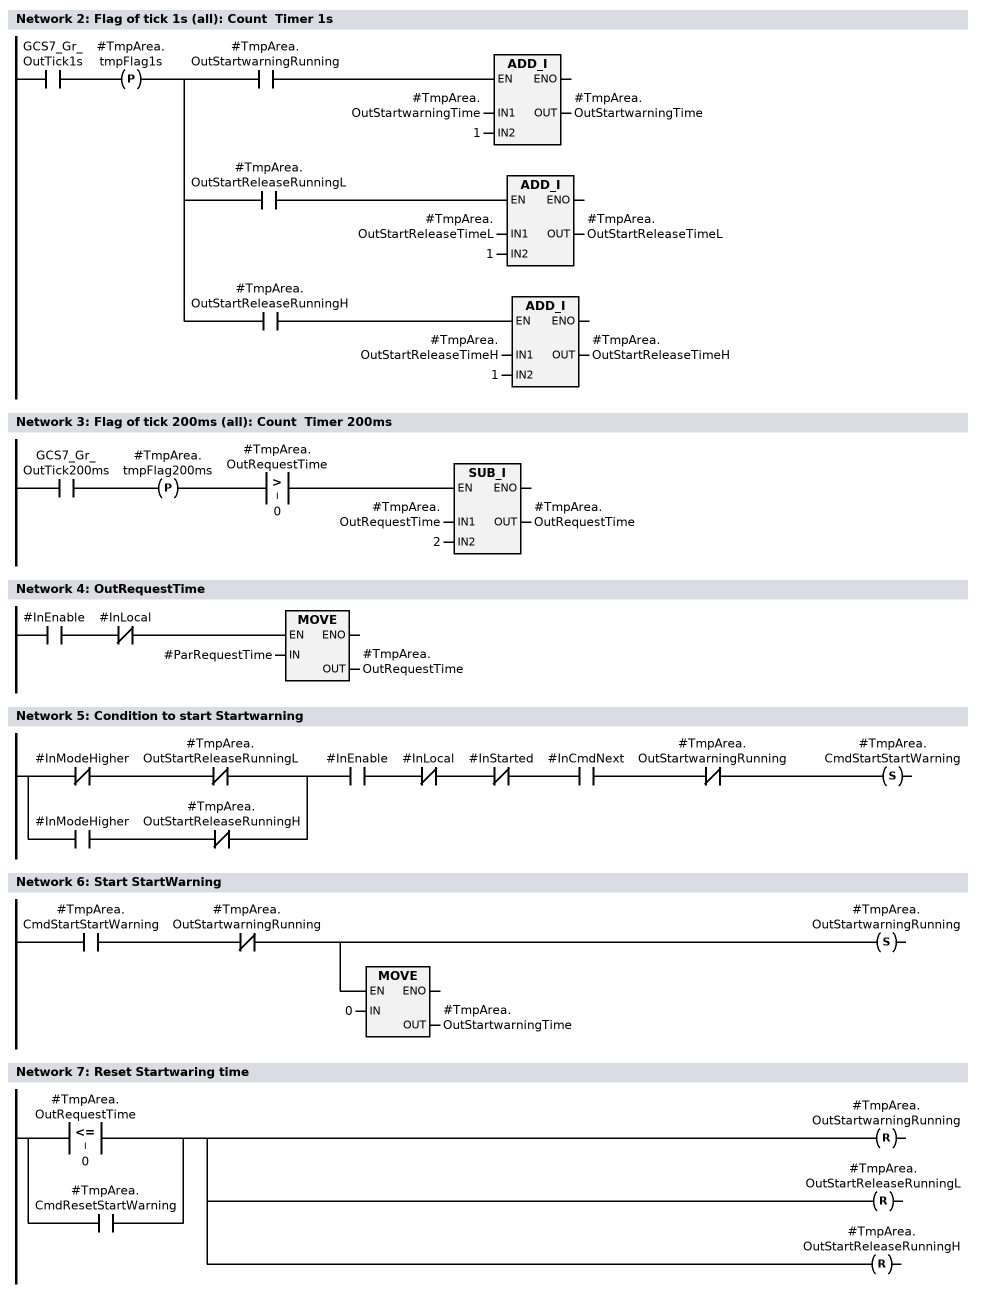
NETWORK
TITLE = Flag of tick 1s (all): Count  Timer 1s
      A     "GCS7_Gr_OutTick1s";	// "Gr.OutTick1s"
      FP    #TmpArea.tmpFlag1s;
      =     L 8.0;
      A     L 8.0;
      A     #TmpArea.OutStartwarningRunning;
      JNB   _001;
      L     #TmpArea.OutStartwarningTime;
      L     1;
      +I;
      T     #TmpArea.OutStartwarningTime;
_001: NOP   0;
      A     L 8.0;
      A     #TmpArea.OutStartReleaseRunningL;
      JNB   _002;
      L     #TmpArea.OutStartReleaseTimeL;
      L     1;
      +I;
      T     #TmpArea.OutStartReleaseTimeL;
_002: NOP   0;
      A     L 8.0;
      A     #TmpArea.OutStartReleaseRunningH;
      JNB   _003;
      L     #TmpArea.OutStartReleaseTimeH;
      L     1;
      +I;
      T     #TmpArea.OutStartReleaseTimeH;
_003: NOP   0;
NETWORK
TITLE = Flag of tick 200ms (all): Count  Timer 200ms
      A     "GCS7_Gr_OutTick200ms";
      FP    #TmpArea.tmpFlag200ms;
      A(;
      L     #TmpArea.OutRequestTime;
      L     0;
      >I;
      );
      JNB   _004;
      L     #TmpArea.OutRequestTime;
      L     2;
      -I;
      T     #TmpArea.OutRequestTime;
_004: NOP   0;
NETWORK
TITLE = OutRequestTime
      A     #InEnable;
      AN    #InLocal;
      JNB   _005;
      L     #ParRequestTime;
      T     #TmpArea.OutRequestTime;
_005: NOP   0;
NETWORK
TITLE = Condition to start Startwarning
//Check if any elementet needs to start
//
      A(;
      AN    #InModeHigher;
      AN    #TmpArea.OutStartReleaseRunningL;
      O;
      A     #InModeHigher;
      AN    #TmpArea.OutStartReleaseRunningH;
      );
      A     #InEnable;
      AN    #InLocal;
      AN    #InStarted;
      A     #InCmdNext;
      AN    #TmpArea.OutStartwarningRunning;
      S     #TmpArea.CmdStartStartWarning;
NETWORK
TITLE = Start StartWarning
      A     #TmpArea.CmdStartStartWarning;
      AN    #TmpArea.OutStartwarningRunning;
      =     L 8.0;
      A     L 8.0;
      BLD   102;
      S     #TmpArea.OutStartwarningRunning;
      A     L 8.0;
      JNB   _006;
      L     0;
      T     #TmpArea.OutStartwarningTime;
_006: NOP   0;
NETWORK
TITLE = Reset Startwaring time
      O(;
      L     #TmpArea.OutRequestTime;
      L     0;
      <=I;
      );
      O     #TmpArea.CmdResetStartWarning;
      R     #TmpArea.OutStartwarningRunning;
      R     #TmpArea.OutStartReleaseRunningL;
      R     #TmpArea.OutStartReleaseRunningH;
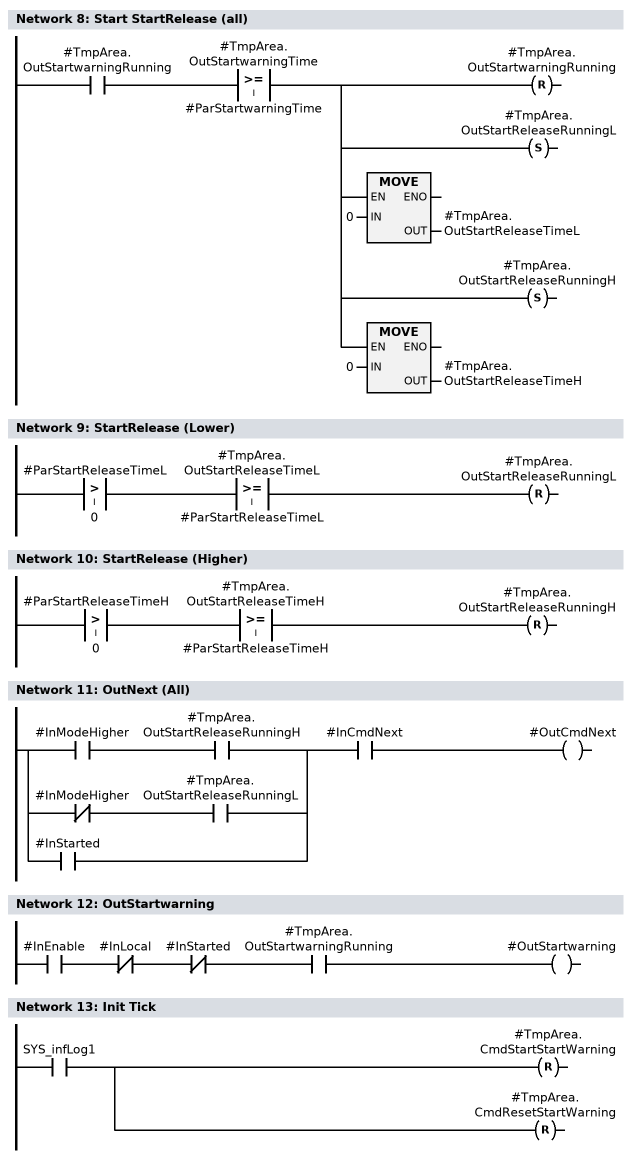
NETWORK
TITLE = Start StartRelease (all)
      A     #TmpArea.OutStartwarningRunning;
      A(;
      L     #TmpArea.OutStartwarningTime;
      L     #ParStartwarningTime;
      >=I;
      );
      =     L 8.0;
      A     L 8.0;
      BLD   102;
      R     #TmpArea.OutStartwarningRunning;
      A     L 8.0;
      BLD   102;
      S     #TmpArea.OutStartReleaseRunningL;
      A     L 8.0;
      JNB   _007;
      L     0;
      T     #TmpArea.OutStartReleaseTimeL;
_007: NOP   0;
      A     L 8.0;
      BLD   102;
      S     #TmpArea.OutStartReleaseRunningH;
      A     L 8.0;
      JNB   _00b;
      L     0;
      T     #TmpArea.OutStartReleaseTimeH;
_00b: NOP   0;
NETWORK
TITLE = StartRelease (Lower)
      A(;
      L     #ParStartReleaseTimeL;
      L     0;
      >I;
      );
      A(;
      L     #TmpArea.OutStartReleaseTimeL;
      L     #ParStartReleaseTimeL;
      >=I;
      );
      R     #TmpArea.OutStartReleaseRunningL;
NETWORK
TITLE = StartRelease (Higher)
      A(;
      L     #ParStartReleaseTimeH;
      L     0;
      >I;
      );
      A(;
      L     #TmpArea.OutStartReleaseTimeH;
      L     #ParStartReleaseTimeH;
      >=I;
      );
      R     #TmpArea.OutStartReleaseRunningH;
NETWORK
TITLE = OutNext (All)
      A(;
      A     #InModeHigher;
      A     #TmpArea.OutStartReleaseRunningH;
      O;
      AN    #InModeHigher;
      A     #TmpArea.OutStartReleaseRunningL;
      O     #InStarted;	//[1.1]
      );
      A     #InCmdNext;
      =     #OutCmdNext;
NETWORK
TITLE = OutStartwarning
      A     #InEnable;
      AN    #InLocal;
      AN    #InStarted;
      A     #TmpArea.OutStartwarningRunning;
      =     #OutStartwarning;
NETWORK
TITLE = Init Tick 
      A     "SYS_infLog1";
      R     #TmpArea.CmdStartStartWarning;
      R     #TmpArea.CmdResetStartWarning;
NETWORK
TITLE = Store Object Data of last warning
      A     #OutStartwarning;
      JNB   _009;
      L     DBNO;
      T     #OutWarningObjectDB;
      L     #InArea;
      T     #OutWarningArea;
_009: NOP   0;
NETWORK
TITLE = Store Area Data
      LAR1  P##TmpArea;
      L     DID [AR1,P#0.0];
      LAR1  #AddrReading;
      T     DID [AR1,P#0.0];
      LAR1  P##TmpArea;
      L     DID [AR1,P#4.0];
      LAR1  #AddrReading;
      T     DID [AR1,P#4.0];
      LAR1  P##TmpArea;
      L     DIW [AR1,P#8.0];
      LAR1  #AddrReading;
      T     DIW [AR1,P#8.0];
END_FUNCTION_BLOCK

